RoboDK station: Continuous-Parts-Conveyor-Infeed.rdk

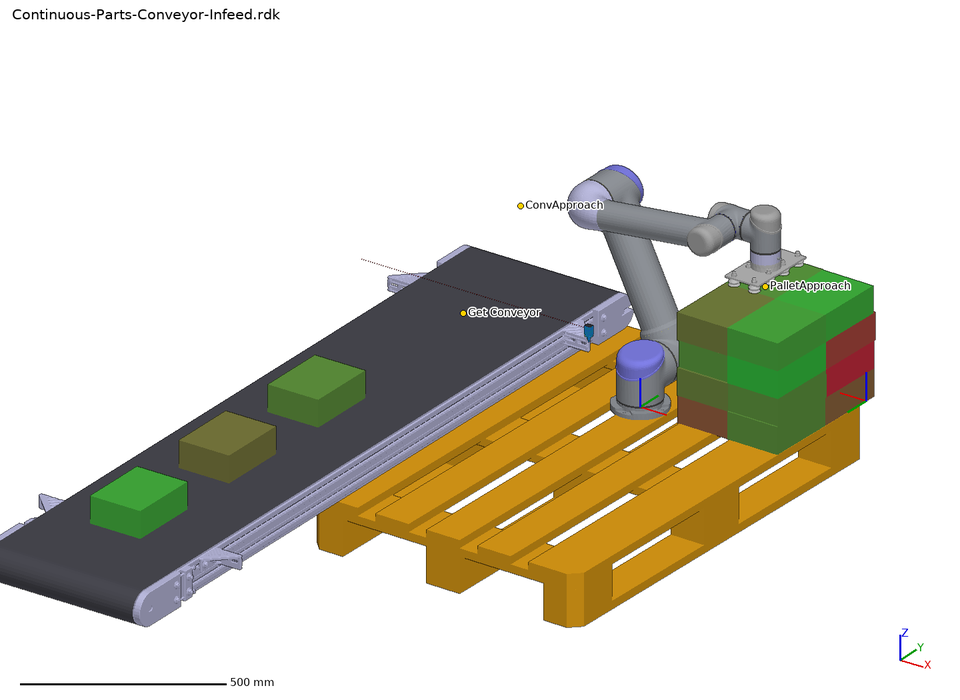
[picture v0: the station drawn from its stored meshes, robots at their saved joint values, targets as dots, program paths as lines]
Station Continuous-Parts-Conveyor-Infeed. Poses are relative to the parent item; angles as X-Y-Z fixed-axis rotations.
Station parameters (name, value as stored): SizeBox, 150, 200, 75, SizePallet, 2,2,4, ConvSpeed, 25.0, SENSOR, 0, parts/min, 4.0
  - frame UR5 Base at (1304.87, 1242.75, -1.35) mm
    - robot UR5: 6 axes, payload 5 kg, reach 850 mm, repeatability 0.1 mm, weight 18.4 kg
        modified DH rows (alpha deg, a mm, theta deg, d mm): 0, 0, 0, 89.2; 90, 0, 180, 0; 0, 425, 0, 0; 0, 392.43, 0, 109; -90, 0, 0, 93.65; 90, 0, 180, 82
        joint limits [-360, -360, -360, -360, -360, -360] to [360, 360, 360, 360, 360, 360]; home [0, -90, 90, 0, 90, 0]; saved at [-180.64, -116.203, 109.647, -83.444, -90, 0]
      - tool Gripper, TCP at (0, 0, 30) mm, rotated rx 0 ry 0 rz 90 deg, size 209.9 x 42 x 100 mm, geometry from test.iges
      - tool TCP, TCP at (0, 0, 67.5) mm, rotated rx 0 ry 0 rz 90 deg
    - target ConvApproach (joint target) at (-414.95, 86.58, 392.2) mm, rotated rx 180 ry 0 rz 0 deg; joints [-26.686, -100.159, 95.166, -85.006, -90, -26.686] of UR5
    - target PalletApproach (joint target) at (297.05, 105.69, 365.83) mm, rotated rx -180 ry 0 rz 179.36 deg; joints [-180.64, -116.203, 109.647, -83.444, -90, 0] of UR5
    - frame Pallet at (419.96, 356.44, -8.51) mm, rotated rx 0 ry 0 rz 179.17 deg
      - object Europallet at (0, 0, 0) mm, size 800 x 144 x 1200 mm, geometry from User Library-Europallet.igs
      - object Part at (75, 69, 37.5) mm, size 150 x 200 x 75 mm, geometry from box.sld
      - object Part at (225, 67, 37.5) mm, size 150 x 200 x 75 mm, geometry from box.sld
      - object Part at (75, 269, 37.5) mm, size 150 x 200 x 75 mm, geometry from box.sld
      - object Part at (225, 267, 37.5) mm, size 150 x 200 x 75 mm, geometry from box.sld
      - object Part at (75, 69, 112.5) mm, size 150 x 200 x 75 mm, geometry from box.sld
      - object Part at (225, 69, 112.5) mm, size 150 x 200 x 75 mm, geometry from box.sld
      - object Part at (75, 265, 112.5) mm, size 150 x 200 x 75 mm, geometry from box.sld
      - object Part at (225, 269, 112.5) mm, size 150 x 200 x 75 mm, geometry from box.sld
      - object Part at (75, 62, 187.5) mm, size 150 x 200 x 75 mm, geometry from box.sld
      - object Part at (225, 65, 187.5) mm, size 150 x 200 x 75 mm, geometry from box.sld
      - object Part at (75, 267, 187.5) mm, size 150 x 200 x 75 mm, geometry from box.sld
      - object Part at (225, 263, 187.5) mm, size 150 x 200 x 75 mm, geometry from box.sld
      - object Part at (75, 71, 262.5) mm, size 150 x 200 x 75 mm, geometry from box.sld
      - object Part at (225, 69, 262.5) mm, size 150 x 200 x 75 mm, geometry from box.sld
      - object Part at (75, 267, 262.5) mm, size 150 x 200 x 75 mm, geometry from box.sld
      - object Part at (225, 269, 262.5) mm, size 150 x 200 x 75 mm, geometry from box.sld
  - frame ConveyorReference at (597.23, -679.82, 119.18) mm
    - robot Conveyor Belt: 1 axes
        modified DH rows (alpha deg, a mm, theta deg, d mm): 0, 0, 0, 0 linear
        base shift (440, 200, 0) mm, rotated rx 0 ry 90 rz 90 deg
        joint limits [-500000] to [500000]; home [0]; saved at [10000]
      - frame MovingRef at (0, 0, 0) mm
        - object Part at (-8921, 240, 37.5) mm, rotated rx 0 ry 0 rz -90 deg, size 150 x 200 x 75 mm, geometry from box.sld
        - object Part at (-9298, 240, 37.5) mm, rotated rx 0 ry 0 rz -90 deg, size 150 x 200 x 75 mm, geometry from box.sld
        - object Part at (-9673, 240, 37.5) mm, rotated rx 0 ry 0 rz -90 deg, size 150 x 200 x 75 mm, geometry from box.sld
    - object box100mm at (200, 300, 0) mm, size 100 x 100 x 100 mm, geometry from box.sld
    - object Sensor SICK WL4S at (551.19, 1928.29, 24.16) mm, rotated rx 90 ry 0 rz 180 deg, size 683.3 x 45.2 x 12.5 mm, geometry from SICK WL4S-3P1330-Order no.1042068 (1).stp
      - Python program WaitForPart (listed below)
      - Python program SensorActivate (listed below)
    - target Get Conveyor (Cartesian target) at (200, 1900, 0) mm, rotated rx -180 ry 0 rz 0 deg; joints [-12.012, -70.873, 123.705, -142.833, -90, -12.012] of UR5
  - Python program SetSimulationParams (listed below)
  - Python program AddPart (listed below)
  - Python program InputParts (listed below)
  - Python program RobotPackParts (listed below)
  - program MainSimulation (3 instructions, listed below)

--- Python program WaitForPart ---
# Type help("robolink") or help("robodk") for more information
# Press F5 to run the script
# Note: you do not need to keep a copy of this file, your python script is saved with the station
from robolink import *    # API to communicate with RoboDK
from robodk import *      # basic matrix operations
RDK = Robolink()

# This script allows to simulate a laser sensor
# that detect the presence of a part in a plane,
# such as a part crossing a laser sensor in a
# conveyor belt

# The script finishes once a part has been detected
# so it works like a WAIT UNTIL function.

# Use a target from the station as a reference plane:
SENSOR_NAME = 'Sensor SICK WL4S'

# Look for parts with the keyword "Part"
PART_KEYWORD = 'Part'

# Update status every 1 ms
RECHECK_PERIOD = 0.001

# Get the sensor and the detection plane
SENSOR = RDK.Item(SENSOR_NAME, ITEM_TYPE_OBJECT)

# Define a function to detect a target
def part_detected(part):
    """Check if a part is in the detection area (proximity of a point to a plane)"""
    if SENSOR.Collision(part) > 0:
        return True
    return False

# Get all object names
all_objects = RDK.ItemList(ITEM_TYPE_OBJECT)

# Get object items in a list (faster) and filter by keyword
check_objects = []
check_objects_names = []
for i in range(len(all_objects)):
    if all_objects[i].count(PART_KEYWORD) > 0:
        check_objects_names.append(all_objects[i])
        check_objects.append(RDK.Item(all_objects[i]))

# Make sure that there are part that we are expecting
nCheck_objects = len(check_objects)
if nCheck_objects == 0:
    raise Exception('No parts to check for. The keyword is %s.' % PICKABLE_OBJECTS_KEYWORD)

# Loop forever until a part is detected by the sensor
part_available = False
while not part_available:
    for i in range(nCheck_objects):
        if part_detected(check_objects[i]):
            print('Part detected: %s' % check_objects_names[i])
            part_available = True
            break

    # Wait some time...
    pause(RECHECK_PERIOD)

print('Program finished')

--- Python program SensorActivate ---
# Type help("robolink") or help("robodk") for more information
# Press F5 to run the script
# Note: you do not need to keep a copy of this file, your python script is saved with the station
from robolink import *    # API to communicate with RoboDK
from robodk import *      # basic matrix operations
RDK = Robolink()

# This script allows to simulate a laser sensor
# that detect the presence of a part in a plane,
# such as a part crossing a laser sensor in a
# conveyor belt

# Use a target from the station as a reference plane:
SENSOR_NAME = 'Sensor SICK WL4S'
SENSOR_VARIABLE = 'SENSOR'

# Look for parts with the keyword "Part"
OBJECTS_REFERENCE = 'MovingRef'
moving_ref = RDK.Item(OBJECTS_REFERENCE, ITEM_TYPE_FRAME)

# Update status every 1 ms
RECHECK_PERIOD = 0.001

# Get the sensor and the detection plane
SENSOR = RDK.Item(SENSOR_NAME, ITEM_TYPE_OBJECT)

# Start delayed as some parts may be deleted
pause(2)

# Loop forever to detect parts
detected_status = -1
while True:
    detected = 0
    for obj in moving_ref.Childs():
        # check if an object has the part keyword and is detected by the laser
        if SENSOR.Collision(obj) > 0:
            detected = 1
            break

    # update the current status of the sensor
    if detected_status != detected:
        detected_status = detected
        RDK.setParam(SENSOR_VARIABLE, detected_status)
        print('Object detected status --> %i' % detected_status)

    # Wait some time...
    pause(RECHECK_PERIOD)

--- Python program SetSimulationParams ---
# Type help("robolink") or help("robodk") for more information
# Press F5 to run the script
# Note: you do not need to keep a copy of this file, your python script is saved with the station
from robolink import *    # API to communicate with RoboDK
from robodk import *      # basic matrix operations


PARAM_SIZE_BOX = 'SizeBox'
PARAM_SIZE_PALLET = 'SizePallet'
PARAM_CONV_SPEED_MM = 'ConvSpeed'

PARAM_PARTS_X_MINUTE = 'parts/min'



RDK = Robolink()

size_box = RDK.getParam(PARAM_SIZE_BOX)
size_pallet = RDK.getParam(PARAM_SIZE_PALLET)
conv_speed = RDK.getParam(PARAM_CONV_SPEED_MM)
parts_x_minute = RDK.getParam(PARAM_PARTS_X_MINUTE)


# ------------------------------------------------------------
size_box_input = mbox('Enter the size of the box in mm [L,W,H]', entry=size_box)
if size_box_input:
    RDK.setParam(PARAM_SIZE_BOX, size_box_input)
else:
    quit()

# ------------------------------------------------------------
size_pallet_input = mbox('Enter the size of the pallet', entry=size_pallet)
if size_pallet_input:
    RDK.setParam(PARAM_SIZE_PALLET, size_pallet_input)
else:
    quit()


# ------------------------------------------------------------
parts_x_minute_entry = mbox('Enter the number of parts per minute', entry=parts_x_minute)
if parts_x_minute_entry:
    RDK.setParam(PARAM_PARTS_X_MINUTE, parts_x_minute_entry)
else:
    quit()

# ------------------------------------------------------------
conv_speed_input = mbox('Enter the speed of the conveyor in mm/s', entry=conv_speed)
if conv_speed_input:
    RDK.setParam(PARAM_CONV_SPEED_MM, conv_speed_input)
    conv_speed = float(conv_speed_input)
    conv = RDK.Item('Conveyor Belt', ITEM_TYPE_ROBOT)
    conv.setSpeed(conv_speed)

else:
    quit()

--- Python program AddPart ---
# Type help("robolink") or help("robodk") for more information
# Press F5 to run the script
# Note: you do not need to keep a copy of this file, your python script is saved with the station
from robolink import *    # API to communicate with RoboDK
from robodk import *      # basic matrix operations
import random
RDK = Robolink()

PART_NAME = 'box100mm'
CONVEYOR_REF = 'MovingRef'

SIZE_BOX = RDK.getParam('SizeBox')

SIZE_BOX_XYZ = [float(x.replace(' ','')) for x in SIZE_BOX.split(',')]
[SIZE_BOX_X, SIZE_BOX_Y, SIZE_BOX_Z] = SIZE_BOX_XYZ

# Create a new part and place it on top of the conveyor, adjusting the height
part = RDK.Item(PART_NAME, ITEM_TYPE_OBJECT)
conveyor_ref = RDK.Item(CONVEYOR_REF, ITEM_TYPE_FRAME)
part_pos = part.PoseAbs()
part.Copy()
newpart = conveyor_ref.Paste()
newpart.setPoseAbs(part_pos*transl(0,0,SIZE_BOX_Z/2))
newpart.setName('Part')
newpart.Scale([SIZE_BOX_X/100, SIZE_BOX_Y/100, SIZE_BOX_Z/100]) #scale with respect to the reference object (100mm cube)
color = random.uniform(0.1 , 0.9)
newpart.Recolor([1-color, color, 0.2, 1]) #set RGBA color
newpart.setVisible(True, False) #make item visible but hide the reference frame

--- Python program InputParts ---
# Type help("robolink") or help("robodk") for more information
# Press F5 to run the script
# Note: you do not need to keep a copy of this file, your python script is saved with the station
from robolink import *    # API to communicate with RoboDK
from robodk import *      # basic matrix operations

# Use RoboDK API as RDK
RDK = Robolink()

PARAM_PARTS_X_MINUTE = 'parts/min'

parts_x_minute = RDK.getParam(PARAM_PARTS_X_MINUTE)

add_part = RDK.Item('AddPart', ITEM_TYPE_PROGRAM_PYTHON)

conv = RDK.Item('Conveyor Belt', ITEM_TYPE_ROBOT)

# turn off rendering (much faster when setting up the station)
#RDK.Render(False)
# cleanup previous simulation (generated parts and tools)
all_objects = RDK.ItemList(ITEM_TYPE_OBJECT, False)
for item in all_objects:
    if item.Name().startswith("Part"):
        item.Delete()

# Turn on rendering
#RDK.Render(True)

conv.setJoints([0])
conv.MoveJ([10000], False)


SECONDS_X_PART = 60.0 / parts_x_minute
tic()
timer_last = toc()
simulation_time = SECONDS_X_PART
while True:
    timer = toc()
    simulation_time = simulation_time + (timer - timer_last) * RDK.SimulationSpeed()
    timer_last = timer
    if simulation_time >= SECONDS_X_PART:
        simulation_time = simulation_time - SECONDS_X_PART
        add_part.RunProgram()

    pause(0.01)

--- Python program RobotPackParts ---
# Type help("robolink") or help("robodk") for more information
# Press F5 to run the script
# Note: you do not need to keep a copy of this file, your python script is saved with the station
from robolink import *    # API to communicate with RoboDK
from robodk import *      # basic matrix operations

# Use RoboDK API as RL
RDK = Robolink()

# define default approach distance
APPROACH = 100
SENSOR_VARIABLE = 'SENSOR' # station variable

# gather robot, tool and reference frames from the station
robot               = RDK.Item('UR5', ITEM_TYPE_ROBOT)
tool                = RDK.Item('Gripper', ITEM_TYPE_TOOL)
tool_tcp            = RDK.Item('TCP', ITEM_TYPE_TOOL)

frame_pallet        = RDK.Item('Pallet', ITEM_TYPE_FRAME)
frame_conv          = RDK.Item('ConveyorReference', ITEM_TYPE_FRAME)
frame_conv_moving   = RDK.Item('MovingRef', ITEM_TYPE_FRAME)

# gather targets
target_pallet_safe = RDK.Item('PalletApproach', ITEM_TYPE_TARGET)
target_conv_safe = RDK.Item('ConvApproach', ITEM_TYPE_TARGET)
target_conv = RDK.Item('Get Conveyor', ITEM_TYPE_TARGET)

# get variable parameters
SIZE_BOX = RDK.getParam('SizeBox')
SIZE_PALLET = RDK.getParam('SizePallet')
SIZE_BOX_XYZ = [float(x.replace(' ','')) for x in SIZE_BOX.split(',')]
SIZE_PALLET_XYZ = [float(x.replace(' ','')) for x in SIZE_PALLET.split(',')]
SIZE_BOX_Z = SIZE_BOX_XYZ[2] # the height of the boxes is important to take into account when approaching the positions

def box_calc(size_xyz, pallet_xyz):
    """Calculates a list of points to store parts in a pallet"""
    [size_x, size_y, size_z] = size_xyz
    [pallet_x, pallet_y, pallet_z] = pallet_xyz
    xyz_list = []
    for h in range(int(pallet_z)):
        for j in range(int(pallet_y)):
            for i in range(int(pallet_x)):
                xyz_list = xyz_list + [[(i+0.5)*size_x, (j+0.5)*size_y, (h+0.5)*size_z]]
    return xyz_list

def TCP_On(toolitem):
    """Attaches the closest object to the toolitem Htool pose,
    It will also output appropriate function calls on the generated robot program (call to TCP_On)"""
    toolitem.AttachClosest()
    toolitem.RDK().RunMessage('Set air valve on')
    toolitem.RDK().RunProgram('TCP_On()')

def TCP_Off(toolitem, itemleave=0):
    """Detaches the closest object attached to the toolitem Htool pose,
    It will also output appropriate function calls on the generated robot program (call to TCP_Off)"""
    #toolitem.DetachClosest(itemleave)
    toolitem.DetachAll(itemleave)
    toolitem.RDK().RunMessage('Set air valve off')
    toolitem.RDK().RunProgram('TCP_Off()')

# calculate an array of positions to get/store the parts
parts_positions = box_calc(SIZE_BOX_XYZ, SIZE_PALLET_XYZ)

# Calculate a new TCP that takes into account the size of the part (targets are set to the center of the box)
tool_xyzrpw = tool.PoseTool()*transl(0,0,SIZE_BOX_Z/2)
tool_tcp.setPoseTool(tool_xyzrpw)
#tool_tcp = robot.AddTool(tool_xyzrpw, 'TCP')

# ---------------------------------------------------------------------------------
# -------------------------- PROGRAM START ----------------------------------------

def WaitSensor():
    if RDK.RunMode() == RUNMODE_SIMULATE:
        # Simulate the sensor by waiting for the SENSOR status to turn to 1 (object present)
        while RDK.getParam(SENSOR_VARIABLE) == 0:
            pause(0.001)
    else:
        RDK.RunProgram('WaitSensor')
    print("Part detected")

robot.setTool(tool_tcp)
nparts = len(parts_positions)
i = 0
while i < nparts:
    # ----------- place the box i on the convegor ------
    # approach to the conveyor
    robot.setFrame(frame_conv)
    target_conv_pose = target_conv.Pose()*transl(0,0,-SIZE_BOX_Z/2)
    target_conv_app = target_conv_pose*transl(0,0,-APPROACH)
    robot.MoveJ(target_conv_safe)
    robot.MoveJ(target_conv_app)
    WaitSensor()
    robot.MoveL(target_conv_pose)
    TCP_On(tool) # detach an place the object in the moving reference frame of the conveyor
    robot.MoveL(target_conv_app)
    robot.MoveJ(target_conv_safe)

    # ----------- take a part from the conveyor ------
    # get the xyz position of part i
    robot.setFrame(frame_pallet)
    part_position_i = parts_positions[i]
    target_i = transl(part_position_i)*rotx(pi)
    target_i_app = target_i * transl(0,0,-(APPROACH+SIZE_BOX_Z))
    # approach to the pallet
    robot.MoveJ(target_pallet_safe)
    # get the box i
    robot.MoveJ(target_i_app)
    robot.MoveL(target_i)
    TCP_Off(tool, frame_pallet) # attach the closest part
    robot.MoveL(target_i_app)
    robot.MoveJ(target_pallet_safe)

    i = i + 1

--- program MainSimulation ---
  Run RobotPackParts
  Run SensorActivate
  Run InputParts
